ABB RobotStudio station: Aufgabe1.rsstnx

Station Aufgabe1 (saved by RobotStudio 23.2.10478.1)
Controller Steuerung1
  mechanical unit ROB_1: IRB140_6_81_C_03, 6 joints, base frame (0, 0, 0) mm
Layout (positions relative to the parent item):
  - IRB140_6_81_C_03 [mechanism, from %ABB.RobotStudio.Models.IRB140%\IRB140_6_81_C_G_03.rslib] at (0, 0, 0) mm; joint values [0.807, -0.7346, 0.8068, -0.5321, 1.0684, 0.9647] (rad or m)
  - MyTool [mechanism, from Training Objects\myTool.rslib] at (183.67, 150, 540.53) mm, rotated rx 180 ry 38 rz 180 deg
  - table_and_fixture_140 [part, from Training Objects\propeller_table.rslib] at (400, -175, 0) mm
  - Koordinatensystem_1 [frame] at (525, -125, 323) mm
Attachment: MyTool is attached to IRB140_6_81_C_03 / Link6
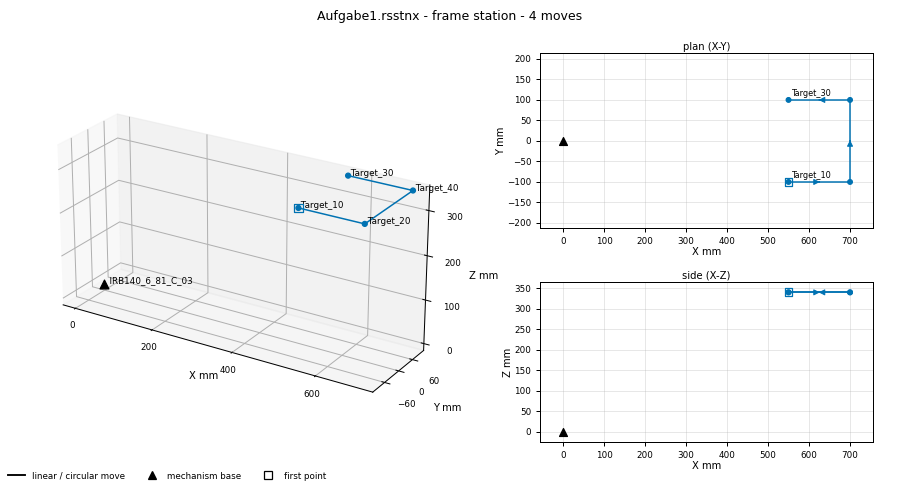
[picture p0: tool path of Aufgabe1.rsstnx in frame station, 4 of 4 moves have a stored position in this frame; points joined in program order, loops and branches not executed]
Targets, tools, work objects and paths stored in the station, written as RAPID:
! task T_ROB1
MODULE CalibData
  PERS tooldata MyTool:=[TRUE,[[31.792631019,0,229.638935148],[0.945518576,0,0.325568154,0]],[1,[0,0,1],[1,0,0,0],0,0,0]];
  TASK PERS wobjdata table:=[FALSE,TRUE,"",[[0,0,0],[1,0,0,0]],[[0,0,0],[1,0,0,0]]];
ENDMODULE

! task T_ROB1
MODULE Module1
  CONST robtarget Target_10:=[[550,-100,340],[0,0,1,0],[-1,0,-1,0],[9E+09,9E+09,9E+09,9E+09,9E+09,9E+09]];
  CONST robtarget Target_20:=[[700,-100,340],[0,0,1,0],[-1,0,-1,0],[9E+09,9E+09,9E+09,9E+09,9E+09,9E+09]];
  CONST robtarget Target_30:=[[550,100,340],[0,0,1,0],[0,-1,0,0],[9E+09,9E+09,9E+09,9E+09,9E+09,9E+09]];
  CONST robtarget Target_40:=[[700,100,340],[0,0,1,0],[0,-1,0,0],[9E+09,9E+09,9E+09,9E+09,9E+09,9E+09]];
  PROC Path_10()
    MoveL Target_10,v1000,z100,MyTool\WObj:=table;
    MoveL Target_20,v100,fine,MyTool\WObj:=table;
    MoveL Target_40,v1000,z100,MyTool\WObj:=table;
    MoveL Target_30,v1000,z100,MyTool\WObj:=table;
  ENDPROC
  PROC main()
    Path_10;
  ENDPROC
ENDMODULE

